Universal Robots PolyScope program: taskboard_retainer_and_nut_v4_hu.urp

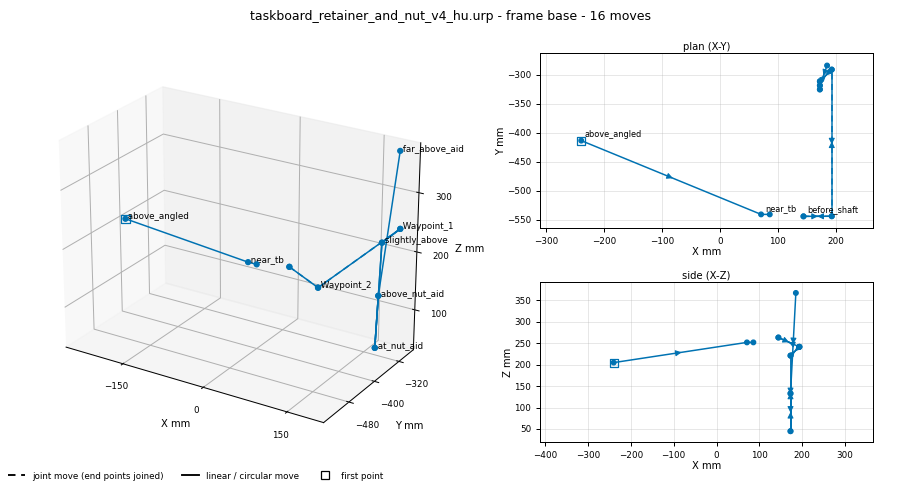
[picture p0: tool path of taskboard_retainer_and_nut_v4_hu.urp in frame base, 16 of 21 moves have a stored position in this frame; points joined in program order, loops and branches not executed]
Program taskboard_retainer_and_nut_v4_hu (installation=default directory=/programs/wrs2020 createdIn=5.6.0.90886 lastSavedIn=5.9.1.1031110 robotSerialNumber=20205500180)
Calibrated DH parameters: a=[0, -0.425, -0.3922, 0, 0, 0]; d=[0.1625, 0, 0, 0.1333, 0.0997, 0.0996]; alpha=[1.570796, 0, 0, 1.570796, -1.570796, 0]; deltaTheta=[0, 0, 0, 0, 0, 0]
Robot Program (runOnlyOnce=true)
  SuppressedNode
    MoveJ speed 180 deg/s, acceleration 150 deg/s^2 (useActiveTCP=false) tcp=gripper_140_tip; feature=Base
      Waypoint home: TCP in base x=133.727 y=-178.735 z=460.339 mm, rx=-0.0013 ry=3.138 rz=0.0408 rad; joints [90.031, -120.136, 80.128, -48.416, -89.757, -0.16] deg; TCP offset x=0 y=0 z=220 mm, rx=0 ry=0 rz=0 rad
  SuppressedNode
    MoveJ speed 180 deg/s, acceleration 150 deg/s^2 (useActiveTCP=true) feature=Base
      Waypoint Waypoint_12: TCP in base x=-82.102 y=-275.549 z=387.348 mm, rx=-0.1814 ry=-3.1114 rz=0.2863 rad; joints [35.849, -127.007, 98.51, -68.6, -82.206, -47.132] deg; TCP offset x=0 y=0 z=220 mm, rx=0 ry=0 rz=0 rad
  SuppressedNode
    URCap Gripper (Robotiq_Grippers, Robotiq Inc.) dataModel(position=44.705882352941174, force=100.0, speed=100.0, positionInDouble=44.705882352941174, forceInDouble=100.0, speedInDouble=100.0, slaveIds=[9], blocking=true)
  SuppressedNode
    MoveJ speed 180 deg/s, acceleration 150 deg/s^2 (useActiveTCP=true) feature=Base
      Waypoint above_idler: TCP in base x=-247.496 y=-411.554 z=147.62 mm, rx=-3.1227 ry=-0.1237 rz=0.0253 rad; joints [43.772, -91.344, 109.218, -107.951, -91.315, 129.235] deg
  SuppressedNode
    MoveL speed 50 mm/s, acceleration 1200 mm/s^2 (useActiveTCP=true) feature=Base
      Waypoint at_pulley_1: motionParameters(jointSpeed=1.047198 jointAcceleration=1.396263 cartesianSpeed=0.5 cartesianAcceleration=1.2); TCP in base x=-247.452 y=-411.527 z=69.357 mm, rx=-3.1227 ry=-0.1238 rz=0.0253 rad; joints [43.775, -86.663, 116.99, -120.4, -91.317, 129.235] deg
  URCap Gripper (Robotiq_Grippers, Robotiq Inc.) dataModel(position=100.0, force=0.0, speed=0.0, positionInDouble=100.0, forceInDouble=0.0, speedInDouble=0.0, slaveIds=[9], blocking=true)
  URCap Gripper (Robotiq_Grippers, Robotiq Inc.) dataModel(position=45.09803921568627, force=0.0, speed=0.0, positionInDouble=45.09803921568627, forceInDouble=0.0, speedInDouble=0.0, slaveIds=[9], blocking=true)
  MoveL speed 800 mm/s, acceleration 1200 mm/s^2 (useActiveTCP=true) feature=Base
    Waypoint turn_right (Relative): relativeFromPosition TCP in base x=-247.464 y=-411.551 z=65.306 mm, rx=2.2244 ry=-2.2171 rz=-0.0361 rad; joints [43.776, -86.348, 117.34, -121.068, -91.317, -136.413] deg; TCP in base x=-247.474 y=-411.554 z=65.268 mm, rx=-0.0035 ry=-3.1247 rz=-0.0244 rad; joints [43.774, -86.343, 117.34, -121.072, -91.315, -46.098] deg
  URCap Gripper (Robotiq_Grippers, Robotiq Inc.) dataModel(position=100.0, force=0.0, speed=0.0, positionInDouble=100.0, forceInDouble=0.0, speedInDouble=0.0, slaveIds=[9], blocking=true)
  URCap Gripper (Robotiq_Grippers, Robotiq Inc.) dataModel(position=57.64705882352941, force=0.0, speed=0.0, positionInDouble=57.64705882352941, forceInDouble=0.0, speedInDouble=0.0, slaveIds=[9], blocking=true)
  MoveL speed 800 mm/s, acceleration 1200 mm/s^2 (useActiveTCP=true) feature=Base
    Waypoint turn_left (Relative): relativeFromPosition TCP in base x=-247.487 y=-411.573 z=65.314 mm, rx=-0.0034 ry=-3.1246 rz=-0.0244 rad; joints [43.776, -86.347, 117.339, -121.073, -91.317, -46.099] deg; TCP in base x=-247.45 y=-411.548 z=65.274 mm, rx=2.2244 ry=-2.2172 rz=-0.0361 rad; joints [43.776, -86.344, 117.339, -121.066, -91.315, -136.41] deg
  MoveL speed 800 mm/s, acceleration 1200 mm/s^2 (useActiveTCP=true) feature=Base
    Waypoint incline (Relative): relativeFromPosition TCP in base x=-240.053 y=-418.618 z=68.067 mm, rx=-3.1413 ry=-0.0077 rz=0.0221 rad; joints [44.528, -86.689, 117.374, -121.253, -90.575, -225.755] deg; TCP in base x=-240.066 y=-413.5 z=66.112 mm, rx=2.4664 ry=-0.0002 rz=-0.0194 rad; joints [17.444, -99.6, 147.461, -152.287, -53.698, -247.795] deg
  URCap Gripper (Robotiq_Grippers, Robotiq Inc.) dataModel(position=100.0, force=0.0, speed=0.0, positionInDouble=100.0, forceInDouble=0.0, speedInDouble=0.0, slaveIds=[9], blocking=true)
  MoveL speed 120 mm/s, acceleration 250 mm/s^2 (useActiveTCP=true) feature=Base
    Waypoint above_angled: motionParameters(jointSpeed=1.047198 jointAcceleration=1.396263 cartesianSpeed=0.25 cartesianAcceleration=1.2); TCP in base x=-239.887 y=-413.598 z=204.833 mm, rx=1.8379 ry=-1.8459 rz=-0.6644 rad; joints [66.077, -97.285, 120.862, -129.87, -125.089, -118.783] deg
    Waypoint near_tb: motionParameters(blendRadius=0.013); TCP in base x=70.932 y=-541.078 z=251.969 mm, rx=-2.2086 ry=1.5312 rz=-1.507 rad; joints [49.874, -97.033, 118.176, -96.847, -32.467, 201.465] deg
    Waypoint in_ridge: motionParameters(jointSpeed=1.047198 jointAcceleration=1.396263 cartesianSpeed=0.02 cartesianAcceleration=1.2); TCP in base x=85.93 y=-541.088 z=251.993 mm, rx=-2.2087 ry=1.5312 rz=-1.507 rad; joints [51.506, -97.754, 119.456, -99.928, -32.098, 204.443] deg
  Popup Message (haltProgram=false message=wait for screw tool to hold inputType=Text)
  URCap Gripper (Robotiq_Grippers, Robotiq Inc.) dataModel(position=41.96078431372549, force=100.0, speed=100.0, positionInDouble=41.96078431372549, forceInDouble=100.0, speedInDouble=100.0, slaveIds=[9], blocking=true)
  MoveL speed 250 mm/s, acceleration 1200 mm/s^2 (useActiveTCP=true) feature=Base
    Waypoint move_away (Relative): relativeFromPosition TCP in base x=81.904 y=-540.987 z=249.22 mm, rx=-2.2078 ry=1.5258 rz=-1.5075 rad; joints [51.039, -97.244, 119.216, -99.021, -32.163, -156.841] deg; TCP in base x=39.536 y=-471.892 z=310.282 mm, rx=-2.2141 ry=1.5067 rz=-1.5033 rad; joints [39.48, -105.154, 112.028, -67.013, -36.755, -177.273] deg
    Waypoint far_above_aid: TCP in base x=185.019 y=-283.793 z=367.304 mm, rx=3.0427 ry=0.0266 rz=0.0843 rad; joints [97.518, -117.381, 97.301, -75.775, -87.414, -173.456] deg
  MoveL speed 250 mm/s, acceleration 1200 mm/s^2 (useActiveTCP=true) feature=Base
    Waypoint above_nut_aid: TCP in base x=172.519 y=-318.273 z=132.878 mm, rx=3.1334 ry=-0.0123 rz=-0.0179 rad; joints [97.626, -109.17, 125.745, -106.863, -90.541, -171.937] deg
    URCap Gripper (Robotiq_Grippers, Robotiq Inc.) dataModel(position=21.96078431372549, force=100.0, speed=100.0, positionInDouble=21.96078431372549, forceInDouble=100.0, speedInDouble=100.0, slaveIds=[9], blocking=true)
    Waypoint at_nut_aid: TCP in base x=172.519 y=-325.105 z=44.86 mm, rx=3.1334 ry=-0.0123 rz=-0.0179 rad; joints [97.451, -101.585, 134.781, -123.486, -90.53, -172.054] deg
    URCap Gripper (Robotiq_Grippers, Robotiq Inc.) dataModel(position=100.0, force=100.0, speed=100.0, positionInDouble=100.0, forceInDouble=100.0, speedInDouble=100.0, slaveIds=[9], blocking=true)
    Waypoint slightly_above: TCP in base x=172.519 y=-311.073 z=221.087 mm, rx=3.1334 ry=-0.0123 rz=-0.0179 rad; joints [97.806, -112.461, 114.667, -92.492, -90.559, -171.799] deg
  MoveL speed 250 mm/s, acceleration 1200 mm/s^2 (useActiveTCP=true) feature=Base
    Waypoint Waypoint_1: TCP in base x=193.098 y=-290.824 z=241.653 mm, rx=-2.26 ry=-2.0992 rz=0.0999 rad; joints [105.872, -111.142, 110.658, -88.291, -94.599, -249.911] deg
    Waypoint Waypoint_2: motionParameters(blendRadius=0.036); TCP in base x=193.098 y=-544.308 z=241.653 mm, rx=-2.26 ry=-2.0992 rz=0.0999 rad; joints [98.952, -79.277, 82.032, -92.106, -94.688, -256.794] deg
    Waypoint before_shaft: TCP in base x=144.251 y=-544.485 z=263.341 mm, rx=2.2425 ry=2.1895 rz=-0.0817 rad; joints [92.3, -83.868, 84.821, -93.226, -91.975, -266.37] deg
  MoveL speed 5 mm/s, acceleration 100 mm/s^2 (useActiveTCP=true) feature=Base
    Waypoint at_shaft (Relative): relativeFromPosition TCP in base x=144.251 y=-544.503 z=263.351 mm, rx=2.2425 ry=2.1895 rz=-0.0818 rad; joints [92.3, -83.867, 84.819, -93.228, -91.976, -266.371] deg; TCP in base x=137.728 y=-544.491 z=263.397 mm, rx=2.2425 ry=2.1895 rz=-0.0819 rad; joints [91.604, -84.12, 85.101, -93.283, -91.949, -267.066] deg
    Popup Message (haltProgram=false message=turn on motor, then press enter to start spiral motion inputType=Text)
    Force Frame feature=Base; selection=[1, 0, 0, 0, 0, 0]; wrench=[-5, 0, 10, 0, 0, 0]; limitsForce=[0.005, 0.15, 0.01, 1.047198, 1.047198, 1.047198]; limitsMotion=[0.1, 0.1, 0.1, 0.349066, 0.349066, 0.349066]
      Loop Counting (count=5) loopVariable(name=Loop_1)
        MoveDirectionNode (selectedDirection=YPlus) feature=Base
          Until DISTANCE (allowActions=false deceleration=3 distanceNodeType=STOP) Distance=0.002; motionParameters(blendRadius=0)
        MoveDirectionNode (selectedDirection=ZPlus) feature=Base
          Until DISTANCE (allowActions=false deceleration=3 distanceNodeType=STOP) Distance=0.002; motionParameters(blendRadius=0)
        MoveDirectionNode (selectedDirection=YMinus) feature=Base
          Until DISTANCE (allowActions=false deceleration=3 distanceNodeType=STOP) Distance=0.002; motionParameters(blendRadius=0)
        MoveDirectionNode (selectedDirection=YMinus) feature=Base
          Until DISTANCE (allowActions=false deceleration=3 distanceNodeType=STOP) Distance=0.002; motionParameters(blendRadius=0)
        MoveDirectionNode (selectedDirection=ZMinus) feature=Base
          Until DISTANCE (allowActions=false deceleration=3 distanceNodeType=STOP) Distance=0.002; motionParameters(blendRadius=0)
        MoveDirectionNode (selectedDirection=YPlus) feature=Base
          Until DISTANCE (allowActions=false deceleration=3 distanceNodeType=STOP) Distance=0.002; motionParameters(blendRadius=0)
        MoveDirectionNode (selectedDirection=YPlus) feature=Base
          Until DISTANCE (allowActions=false deceleration=3 distanceNodeType=STOP) Distance=0.002; motionParameters(blendRadius=0)
        MoveDirectionNode (selectedDirection=ZMinus) feature=Base
          Until DISTANCE (allowActions=false deceleration=3 distanceNodeType=STOP) Distance=0.002; motionParameters(blendRadius=0)
        MoveDirectionNode (selectedDirection=YMinus) feature=Base
          Until DISTANCE (allowActions=false deceleration=3 distanceNodeType=STOP) Distance=0.002; motionParameters(blendRadius=0)
        MoveDirectionNode (selectedDirection=YMinus) feature=Base
          Until DISTANCE (allowActions=false deceleration=3 distanceNodeType=STOP) Distance=0.002; motionParameters(blendRadius=0)
        MoveDirectionNode (selectedDirection=ZPlus) feature=Base
          Until DISTANCE (allowActions=false deceleration=3 distanceNodeType=STOP) Distance=0.002; motionParameters(blendRadius=0)
        MoveDirectionNode (selectedDirection=YPlus) feature=Base
          Until DISTANCE (allowActions=false deceleration=3 distanceNodeType=STOP) Distance=0.002; motionParameters(blendRadius=0)
  Popup Message (haltProgram=false message=ok? inputType=Text)
  MoveJ speed 60 deg/s, acceleration 80 deg/s^2 (useActiveTCP=true) feature=Base
    Waypoint before_shaft: motionParameters(jointSpeed=1.047198 jointAcceleration=1.396263 cartesianSpeed=0.25 cartesianAcceleration=1.2); TCP in base x=144.251 y=-544.485 z=263.341 mm, rx=2.2425 ry=2.1895 rz=-0.0817 rad; joints [92.3, -83.868, 84.821, -93.226, -91.975, -266.37] deg
    Waypoint Waypoint_2: motionParameters(jointSpeed=2.094395 jointAcceleration=2.094395 cartesianSpeed=0.25 cartesianAcceleration=1.2 blendRadius=0.05); TCP in base x=193.098 y=-544.308 z=241.653 mm, rx=-2.26 ry=-2.0992 rz=0.0999 rad; joints [98.952, -79.277, 82.032, -92.106, -94.688, -256.794] deg
    Waypoint Waypoint_1: motionParameters(jointSpeed=2.094395 jointAcceleration=2.094395 cartesianSpeed=0.25 cartesianAcceleration=1.2); TCP in base x=193.098 y=-290.824 z=241.653 mm, rx=-2.26 ry=-2.0992 rz=0.0999 rad; joints [105.872, -111.142, 110.658, -88.291, -94.599, -249.911] deg
  MoveL speed 250 mm/s, acceleration 1200 mm/s^2 (useActiveTCP=true) feature=Base
    Waypoint slightly_above: TCP in base x=172.519 y=-311.073 z=221.087 mm, rx=3.1334 ry=-0.0123 rz=-0.0179 rad; joints [97.806, -112.461, 114.667, -92.492, -90.559, -171.799] deg
    Waypoint at_nut_aid: TCP in base x=172.519 y=-325.105 z=44.86 mm, rx=3.1334 ry=-0.0123 rz=-0.0179 rad; joints [97.451, -101.585, 134.781, -123.486, -90.53, -172.054] deg
    URCap Gripper (Robotiq_Grippers, Robotiq Inc.) dataModel(position=21.96078431372549, force=100.0, speed=100.0, positionInDouble=21.96078431372549, forceInDouble=100.0, speedInDouble=100.0, slaveIds=[9], blocking=true)
    Waypoint above_nut_aid: TCP in base x=172.519 y=-318.273 z=132.878 mm, rx=3.1334 ry=-0.0123 rz=-0.0179 rad; joints [97.626, -109.17, 125.745, -106.863, -90.541, -171.937] deg
